// TIA Portal V18 export
DATA_BLOCK "LightBarrier_DB"   // DB74
VERSION : 0.1
// stored: AutoNumber true, DBAccessibleFromOPCUA true, InstanceOfName LightBarrier, InstanceOfType FB
"LightBarrier"
   // VAR_INPUT
   //    barrier_ok : Bool;
   // END_VAR
BEGIN
END_DATA_BLOCK
